Yaskawa INFORM job: SYS_CHECK_VACUUM.JBI

/JOB
//NAME SYS_CHECK_VACUUM
//POS
///NPOS 0,0,0,0,0,0
//INST
///DATE 2022/01/20 14:38
///ATTR SC,RW
///GROUP1 RB1
NOP
WAIT T=0.50
IFTHENEXP IN#(2)=OFF
	 SETUALM 8000 "INSUFFICIENT VACUUM DETECTED" 0
ENDIF
END
